// TIA Portal V20 export
TYPE "HMIAxisCtrl_typeInputs"
TITLE = HMIAxisCtrl_typeInputs
// Support: tech.team.motioncontrol@siemens.com 
// Fax: +49 (0) 9131/98-1297
   STRUCT
      enable : Bool;   // TRUE: Enable functionality of FB
      enableAxis : Bool;   // TRUE: Set axis enable; FALSE: Remove axis enable
      resetAxis : Bool;   // Rising edge: Acknowledgement of technology alarms or restart of the axis (depending on configuration)
      jogForward : Bool;   // Rising edge: Move an axis in jog mode (forward); Falling edge: Stop jogging
      jogBackward : Bool;   // Rising edge: Move an axis in jog mode (backward); Falling edge: Stop jogging
      moveVelocity : Bool;   // Rising edge: Move an axis at constant velocity/speed
      stop : Bool;   // Rising edge: Brake an axis until it comes to a standstill
      fastStop : Bool;   // Rising edge: Brake an axis until it comes to a standstill (with fastStop dynamics)
      torqueLimiting : Bool;   // TRUE: Enable force/torque limiting
      homing : Bool;   // Rising edge: Home axis
      posRelative : Bool;   // Rising edge: Move an axis relative to its position when execution of the job began
      posAbsolute : Bool;   // Rising edge: Move an axis to an absolute position
      posSuperimposed : Bool;   // Rising edge: Start a superimposed positioning
      gearInRelative : Bool;   // Rising edge: Start a gearing operation (relative)
      gearInAbsolute : Bool;   // Rising edge: Start a gearing operation (absolute)
      camIn : Bool;   // Rising edge: Start a camming operation
      phasing : Bool;   // Rising edge: Start a phasing operation
      openBrake : Bool;   // TRUE: Open holding brake
   END_STRUCT;
END_TYPE
